{attribute addProperty BoxType "EKM1101-0000-0016"}
{attribute addProperty Id "ErrorBIT10.1251UnderrangeBIT10.1252OverrangeBIT10.1253DiagBIT10.1254Sensor_OvrBIT10.1255OverrunBIT10.1256TxPDO_StateBIT10.12515"}
{attribute addProperty CRC "1725206741"}
{attribute addProperty SizeInBites "16"}
{attribute addProperty SizeInBytes "2"}
TYPE Status_66D490D5 :
STRUCT
	{attribute addProperty Name "Error"}
	Error : BIT;
	{attribute addProperty Name "Underrange"}
	Underrange : BIT;
	{attribute addProperty Name "Overrange"}
	Overrange : BIT;
	{attribute addProperty Name "Diag"}
	Diag : BIT;
	{attribute addProperty Name "Sensor_Ovr"}
	Sensor_Ovr : BIT;
	{attribute addProperty Name "Overrun"}
	Overrun : BIT;
	{attribute 'hide'}
	reserve_1 : BYTE;
	{attribute addProperty Name "TxPDO_State"}
	TxPDO_State : BIT;
	{attribute 'hide'}
	reserve_2 : BIT;
END_STRUCT
END_TYPE

(* stored: Version 1.2.0.0, ProductVersion 3.1.4024.9
   DUT Status_66D490D5: Id {c1e08cb7-1b0e-4e02-b94f-ba12cf9ff2b1} *)
